FUNCTION_BLOCK MockDisposableDeserializer IMPLEMENTS I_Deserializer
VAR
	disposedFlag : BOOL;
END_VAR

METHOD PUBLIC Dispose
VAR_INPUT
END_VAR
disposedFlag := TRUE;
END_METHOD

METHOD GetArray : I_Deserializer
VAR_INPUT
END_VAR
END_METHOD

METHOD GetElementByIndex : I_Deserializer
VAR_INPUT
	Index : UDINT;
END_VAR
END_METHOD

METHOD GetKey : I_Deserializer
VAR_INPUT
	Key : T_MAXSTRING;
END_VAR
END_METHOD

METHOD GetKeyArray : I_Deserializer
VAR_INPUT
	Key : T_MAXSTRING;
END_VAR
END_METHOD

PROPERTY PUBLIC IsDisposed : BOOL
GET
IsDisposed := disposedFlag;
END_GET
END_PROPERTY

METHOD TryDeserializeKeyToObject : BOOL
VAR_INPUT
	Key : T_MAXSTRING;
	Object : I_Deserializable;
END_VAR
END_METHOD

METHOD TryDeserializeToObject : BOOL
VAR_INPUT
	Object : I_Deserializable;
END_VAR
END_METHOD

METHOD TryGetBase64 : BOOL
VAR_INPUT
	pBytes : POINTER TO BYTE;
	nBytes : DINT;
END_VAR
END_METHOD

METHOD TryGetBool : BOOL
VAR_INPUT
	Destination : REFERENCE TO BOOL;
END_VAR
END_METHOD

METHOD TryGetByte : BOOL
VAR_INPUT
	Destination : REFERENCE TO BYTE;
END_VAR
END_METHOD

METHOD TryGetDateTime : BOOL
VAR_INPUT
	Destination : REFERENCE TO DATE_AND_TIME;
END_VAR
END_METHOD

METHOD TryGetDcTime : BOOL
VAR_INPUT
	Destination : REFERENCE TO DCTIME;
END_VAR
END_METHOD

METHOD TryGetDint : BOOL
VAR_INPUT
	Destination : REFERENCE TO DINT;
END_VAR
END_METHOD

METHOD TryGetDword : BOOL
VAR_INPUT
	Destination : REFERENCE TO DWORD;
END_VAR
END_METHOD

METHOD TryGetFileTime : BOOL
VAR_INPUT
	Destination : REFERENCE TO FILETIME;
END_VAR
END_METHOD

METHOD TryGetHexAsBytes : BOOL
VAR_INPUT
	pBytes : POINTER TO BYTE;
	nBytes : DINT;
END_VAR
END_METHOD

METHOD TryGetInt : BOOL
VAR_INPUT
	Destination : REFERENCE TO INT;
END_VAR
END_METHOD

METHOD TryGetKeyBase64 : BOOL
VAR_INPUT
	Key : T_MAXSTRING;
	pBytes : POINTER TO BYTE;
	nBytes : DINT;
END_VAR
END_METHOD

METHOD TryGetKeyBool : BOOL
VAR_INPUT
	Key : T_MAXSTRING;
	Destination : REFERENCE TO BOOL;
END_VAR
END_METHOD

METHOD TryGetKeyByte : BOOL
VAR_INPUT
	Key : T_MAXSTRING;
	Destination : REFERENCE TO BYTE;
END_VAR
END_METHOD

METHOD TryGetKeyDateTime : BOOL
VAR_INPUT
	Key : T_MAXSTRING;
	Destination : REFERENCE TO DATE_AND_TIME;
END_VAR
END_METHOD

METHOD TryGetKeyDcTime : BOOL
VAR_INPUT
	Key : T_MAXSTRING;
	Destination : REFERENCE TO DCTIME;
END_VAR
END_METHOD

METHOD TryGetKeyDint : BOOL
VAR_INPUT
	Key : T_MAXSTRING;
	Destination : REFERENCE TO DINT;
END_VAR
END_METHOD

METHOD TryGetKeyDword : BOOL
VAR_INPUT
	Key : T_MAXSTRING;
	Destination : REFERENCE TO DWORD;
END_VAR
END_METHOD

METHOD TryGetKeyFileTime : BOOL
VAR_INPUT
	Key : T_MAXSTRING;
	Destination : REFERENCE TO FILETIME;
END_VAR
END_METHOD

METHOD TryGetKeyHexAsBytes : BOOL
VAR_INPUT
	Key : T_MAXSTRING;
	pBytes : POINTER TO BYTE;
	nBytes : DINT;
END_VAR
END_METHOD

METHOD TryGetKeyInt : BOOL
VAR_INPUT
	Key : T_MAXSTRING;
	Destination : REFERENCE TO INT;
END_VAR
END_METHOD

METHOD TryGetKeyLint : BOOL
VAR_INPUT
	Key : T_MAXSTRING;
	Destination : REFERENCE TO LINT;
END_VAR
END_METHOD

METHOD TryGetKeyLreal : BOOL
VAR_INPUT
	Key : T_MAXSTRING;
	Destination : REFERENCE TO LREAL;
END_VAR
END_METHOD

METHOD TryGetKeyLtime : BOOL
VAR_INPUT
	Key : T_MAXSTRING;
	Destination : REFERENCE TO LTIME;
END_VAR
END_METHOD

METHOD TryGetKeyLword : BOOL
VAR_INPUT
	Key : T_MAXSTRING;
	Destination : REFERENCE TO LWORD;
END_VAR
END_METHOD

METHOD TryGetKeyReal : BOOL
VAR_INPUT
	Key : T_MAXSTRING;
	Destination : REFERENCE TO REAL;
END_VAR
END_METHOD

METHOD TryGetKeySint : BOOL
VAR_INPUT
	Key : T_MAXSTRING;
	Destination : REFERENCE TO SINT;
END_VAR
END_METHOD

METHOD TryGetKeyString : BOOL
VAR_INPUT
	Key : T_MAXSTRING;
	Destination : REFERENCE TO STRING;
END_VAR
END_METHOD

METHOD TryGetKeyTime : BOOL
VAR_INPUT
	Key : T_MAXSTRING;
	Destination : REFERENCE TO TIME;
END_VAR
END_METHOD

METHOD TryGetKeyTod : BOOL
VAR_INPUT
	Key : T_MAXSTRING;
	Destination : REFERENCE TO TOD;
END_VAR
END_METHOD

METHOD TryGetKeyUdint : BOOL
VAR_INPUT
	Key : T_MAXSTRING;
	Destination : REFERENCE TO UDINT;
END_VAR
END_METHOD

METHOD TryGetKeyUint : BOOL
VAR_INPUT
	Key : T_MAXSTRING;
	Destination : REFERENCE TO UINT;
END_VAR
END_METHOD

METHOD TryGetKeyUlint : BOOL
VAR_INPUT
	Key : T_MAXSTRING;
	Destination : REFERENCE TO ULINT;
END_VAR
END_METHOD

METHOD TryGetKeyUsint : BOOL
VAR_INPUT
	Key : T_MAXSTRING;
	Destination : REFERENCE TO USINT;
END_VAR
END_METHOD

METHOD TryGetKeyWord : BOOL
VAR_INPUT
	Key : T_MAXSTRING;
	Destination : REFERENCE TO WORD;
END_VAR
END_METHOD

METHOD TryGetLint : BOOL
VAR_INPUT
	Destination : REFERENCE TO LINT;
END_VAR
END_METHOD

METHOD TryGetLreal : BOOL
VAR_INPUT
	Destination : REFERENCE TO LREAL;
END_VAR
END_METHOD

METHOD TryGetLtime : BOOL
VAR_INPUT
	Destination : REFERENCE TO LTIME;
END_VAR
END_METHOD

METHOD TryGetLword : BOOL
VAR_INPUT
	Destination : REFERENCE TO LWORD;
END_VAR
END_METHOD

METHOD TryGetReal : BOOL
VAR_INPUT
	Destination : REFERENCE TO REAL;
END_VAR
END_METHOD

METHOD TryGetSint : BOOL
VAR_INPUT
	Destination : REFERENCE TO SINT;
END_VAR
END_METHOD

METHOD TryGetString : BOOL
VAR_INPUT
	Destination : REFERENCE TO STRING;
END_VAR
END_METHOD

METHOD TryGetTime : BOOL
VAR_INPUT
	Destination : REFERENCE TO TIME;
END_VAR
END_METHOD

METHOD TryGetTod : BOOL
VAR_INPUT
	Destination : REFERENCE TO TOD;
END_VAR
END_METHOD

METHOD TryGetUdint : BOOL
VAR_INPUT
	Destination : REFERENCE TO UDINT;
END_VAR
END_METHOD

METHOD TryGetUint : BOOL
VAR_INPUT
	Destination : REFERENCE TO UINT;
END_VAR
END_METHOD

METHOD TryGetUlint : BOOL
VAR_INPUT
	Destination : REFERENCE TO ULINT;
END_VAR
END_METHOD

METHOD TryGetUsint : BOOL
VAR_INPUT
	Destination : REFERENCE TO USINT;
END_VAR
END_METHOD

METHOD TryGetWord : BOOL
VAR_INPUT
	Destination : REFERENCE TO WORD;
END_VAR
END_METHOD

END_FUNCTION_BLOCK

(* stored: Version 1.1.0.1, ProductVersion 3.1.4024.12
   POU MockDisposableDeserializer: Id {21ef6294-d236-02ff-36c4-1ede30b4ee2e}, SpecialFunc None
   Method Dispose: Id {92caf2b9-f081-0528-0e8d-857606ffd3d1}
   Method GetArray: Id {f6b2f126-4ca1-0f9f-0780-ab5c5ac6f498}
   Method GetElementByIndex: Id {3f652932-bf8d-00a4-3a58-3f797c3c9afc}
   Method GetKey: Id {e69a0eb5-6df8-01fd-1874-df010f2cf837}
   Method GetKeyArray: Id {47167e86-9154-0dfd-3f50-fff0db56fead}
   Property IsDisposed: Id {4e3ddbd4-85e0-02a4-36b9-d73d5f448399}
   Get Get: Id {7d635d94-30fd-0cb7-2f56-1c60b357afca}
   Method TryDeserializeKeyToObject: Id {3bf8532c-5862-054b-1f0e-8c4449b91a92}
   Method TryDeserializeToObject: Id {bd5d60c8-c8c2-0061-2023-b563e7215d93}
   Method TryGetBase64: Id {3caf7798-d301-0947-3f47-b5d39e303e66}
   Method TryGetBool: Id {31638b59-2542-0f1f-3357-7193e1f3abe2}
   Method TryGetByte: Id {e4a2d811-e062-0e32-2b79-b56d947f790b}
   Method TryGetDateTime: Id {fede0a76-38e6-0db8-11ea-130b0923471f}
   Method TryGetDcTime: Id {d0146503-4ce3-03f3-28f9-b1bf6780b1fe}
   Method TryGetDint: Id {b9f1a939-5de8-0c7a-050b-408488135aee}
   Method TryGetDword: Id {8cb40e7a-f073-07c3-2cb5-0c13c9af0257}
   Method TryGetFileTime: Id {ede29f83-1b0d-021b-3fca-7ddda4c5e30f}
   Method TryGetHexAsBytes: Id {2ca3d0eb-36bf-0ab3-0370-3d073d9277f5}
   Method TryGetInt: Id {6472c3f7-d94b-0d52-1a4b-b912ecba4591}
   Method TryGetKeyBase64: Id {f7080887-dd42-04a5-37b0-251009065e7b}
   Method TryGetKeyBool: Id {6980de9d-5e4b-03a9-20af-9756cf573ec2}
   Method TryGetKeyByte: Id {d1b0c085-2508-094b-3b8e-0179539501db}
   Method TryGetKeyDateTime: Id {35a03e23-ce55-0a9c-3a4e-58214fac28b6}
   Method TryGetKeyDcTime: Id {1baa76a8-71ec-0d69-3627-fdf6c3d0d9b7}
   Method TryGetKeyDint: Id {97bffc58-f679-0331-1b11-f0ec0d604a5b}
   Method TryGetKeyDword: Id {a7e07a82-9d35-0efd-2537-5a0cbddc80ac}
   Method TryGetKeyFileTime: Id {3b900536-3d28-09ae-0f25-d0a9dbd32177}
   Method TryGetKeyHexAsBytes: Id {028b90bc-37d8-0ecb-10a2-648fa5fd08a0}
   Method TryGetKeyInt: Id {8ee4c5c3-a67a-07cf-2059-03d3a552600f}
   Method TryGetKeyLint: Id {647185d4-1dc8-0e4e-2f17-f0cc753d3b47}
   Method TryGetKeyLreal: Id {fadd976c-302c-0c88-3d7e-790a9097410b}
   Method TryGetKeyLtime: Id {5b22fc71-a24e-0773-327f-7a490e97e8cd}
   Method TryGetKeyLword: Id {ae0bd34d-4b52-03cc-0a00-b01e382837b1}
   Method TryGetKeyReal: Id {f9e96312-3ece-0713-0a44-85c330c42ec1}
   Method TryGetKeySint: Id {dd3f9858-60f5-0ca8-183d-ea41e44eb31a}
   Method TryGetKeyString: Id {970f7651-3123-04c7-19ad-655e7f716147}
   Method TryGetKeyTime: Id {4dca384e-56ab-044d-39a1-f65ff8d43257}
   Method TryGetKeyTod: Id {4ef6563a-5bf6-0e41-09b5-401b6d39da99}
   Method TryGetKeyUdint: Id {6ff878b3-b0ad-0160-223c-cf08238b940d}
   Method TryGetKeyUint: Id {af7b64bd-b397-018a-39df-9df75b56f7bc}
   Method TryGetKeyUlint: Id {3bd97f7d-c41a-0577-3e78-b409be583b5d}
   Method TryGetKeyUsint: Id {a947dbb3-bf33-0b45-3285-d74c75f914ad}
   Method TryGetKeyWord: Id {058db9f5-046b-0aae-2a80-d1c77cda4f7f}
   Method TryGetLint: Id {d47ab359-55d5-0296-29b0-44be8e27ee7a}
   Method TryGetLreal: Id {818e5cd7-21e5-0a0a-12fc-912927c507ed}
   Method TryGetLtime: Id {0473fe2c-591a-0006-2667-61a21b1d8cba}
   Method TryGetLword: Id {dabc8531-7f53-0662-1578-4c62dafbaac3}
   Method TryGetReal: Id {42c3f14e-0f98-0246-24fb-f7c2a317ea74}
   Method TryGetSint: Id {b21bbb98-8b7e-055c-2785-a86c71230c55}
   Method TryGetString: Id {4b8433bf-92ac-05f4-37ce-7ba2c14c58e7}
   Method TryGetTime: Id {20835ca1-f090-0e39-3629-6abb477bb604}
   Method TryGetTod: Id {a4c79a7e-1562-0ce2-1582-ed4a11e6a155}
   Method TryGetUdint: Id {81afa980-1003-0c17-1b7d-014232e8ba51}
   Method TryGetUint: Id {9f44d275-61eb-0de8-21ed-17cefe0ba707}
   Method TryGetUlint: Id {f92f0db9-57ed-03c3-2739-2dfc95b81f84}
   Method TryGetUsint: Id {f987f05a-25bc-0311-3cd8-b97e7dfa66ea}
   Method TryGetWord: Id {88f80eeb-f765-02f2-0aa4-ac4f40c04b45} *)
